FUNCTION_BLOCK stopper (* Tamplate for a simple Basic Function Block Type *)
  (* Standard: 61499-2 *)
  (* Version 0.0, 2018-01-17, 4DIAC-IDE, 4DIAC-Consortium *)
  (* Version 1.0, 2016-05-26, AZ, fortiss GmbH *)
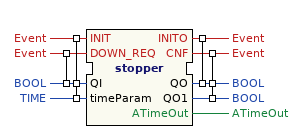
  EVENT_INPUT
    INIT WITH QI, timeParam; (* Initialization Request *)
    DOWN_REQ WITH QI; (* Normal Execution Request *)
  END_EVENT
  EVENT_OUTPUT
    INITO WITH QO; (* Initialization Confirm *)
    CNF WITH QO1, QO; (* Execution Confirmation *)
  END_EVENT
  VAR_INPUT
    QI : BOOL; (* Input event qualifier *)
    timeParam : TIME; (* For timedelay *)
  END_VAR
  VAR_OUTPUT
    QO : BOOL; (* Output event qualifier *)
    QO1 : BOOL;
  END_VAR
  PLUGS
    ATimeOut : ATimeOut;
  END_PLUGS
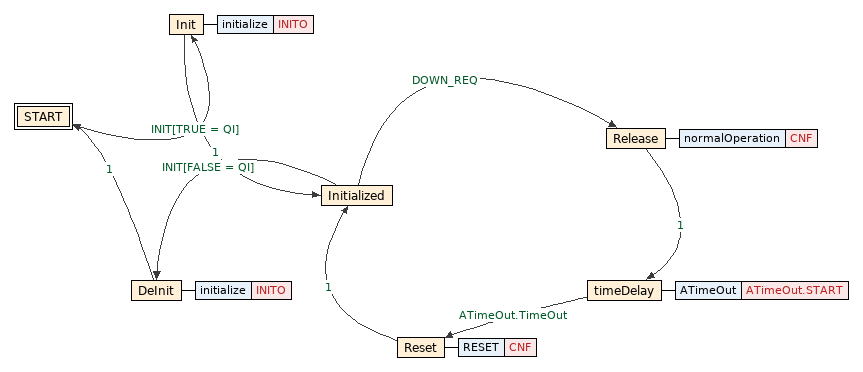
  EC_STATES
    START; (* Initial State *)
    Init : initialize -> INITO; (* Initialization *)
    Release : normalOperation -> CNF; (* Normal execution *)
    Initialized;
    DeInit : initialize -> INITO;
    timeDelay : ATimeOut -> ATimeOut.START; (* After timePara s *)
    Reset : RESET -> CNF;
  END_STATES
  EC_TRANSITIONS
    START TO Init := INIT[TRUE = QI];
    Init TO Initialized := 1;
    Initialized TO Release := DOWN_REQ;
    DeInit TO START := 1;
    Initialized TO DeInit := INIT[FALSE = QI];
    Release TO timeDelay := 1;
    timeDelay TO Reset := ATimeOut.TimeOut;
    Reset TO Initialized := 1;
  END_TRANSITIONS
  ALGORITHM initialize IN ST: (* Initialization algorithm *)
QO := QI;
QO1:=FALSE;
  END_ALGORITHM
  ALGORITHM deInitialize IN ST: (* Normally executed algorithm *)
QO := FALSE;
QO1:=FALSE;
  END_ALGORITHM
  ALGORITHM normalOperation IN ST: (* new algorithm *)
QO1:= true;
  END_ALGORITHM
  ALGORITHM ATimeOut IN ST: (* new algorithm *)
ATimeOut.DT := timeParam;
  END_ALGORITHM
  ALGORITHM RESET IN ST: (* new algorithm *)
QO1:=FALSE;
  END_ALGORITHM
END_FUNCTION_BLOCK
